(* Logix 5000 project; controller DIMTER vendor 1 type 14 code 77 rev 15.4; software revision 15.01; part 3 of 4 *)
(* tags used below, declared in another part *)
   ChainEjectorRunHourTimer : TIMER;   // Chain Ejector Run Hourmeter 1/10th Hour Timer
   CrossBelt1RunHourTimer : TIMER;   // Cross Belt 1 Run Hourmeter 1/10th Hour Timer
   CrossBelt2RunHourTimer : TIMER;   // Cross Belt 2 Run Hourmeter 1/10th Hour Timer
   CrossFeed1RunHourTimer : TIMER;   // Cross Feed 1 Run Hourmeter 1/10th Hour Timer
   CrossFeed2RunHourTimer : TIMER;   // Cross Feed 2 Run Hourmeter 1/10th Hour Timer
   DisplaySplashScreen : BOOL;
   F : BOOL[2016];   // Flags
   FlagTransferIndex : DINT;   // Index Register For Copying Flags to HMI Files
   FlagTransferIndex2 : DINT;
   FLASHER : TIMER;   // Lamp Flasher
   FLASHERB : TIMER;   // Lamp Flasher Reset
   RecordPieceSaw1 : BOOL;   // Record Piece Count For Shift Total
   RecordPieceSaw2 : BOOL;   // Record Piece Count For Shift Total
   Rollcase1RunHourTimer : TIMER;   // Rollcase 1 Run Hourmeter 1/10th Hour Timer
   Rollcase2RunHourTimer : TIMER;   // Rollcase 2 Run Hourmeter 1/10th Hour Timer
   Saw1RunHourTimer : TIMER;   // Saw 1 Run Hourmeter 1/10th Hour Timer
   Saw2RunHourTimer : TIMER;   // Saw 2 Run Hourmeter 1/10th Hour Timer
   SplashScreen : TIMER;
   T : TIMER[100];   // Timers
   WasteBelt1RunHourTimer : TIMER;   // Waste Belt 1 Run Hourmeter 1/10th Hour Timer
   WasteBelt2RunHourTimer : TIMER;   // Waste Belt 2 Run Hourmeter 1/10th Hour Timer
   A122 : ALIAS FOR Local:4:O.Data.2;   // O:4.0/2 A12.2 Reset Failure
   A123 : ALIAS FOR Local:4:O.Data.3;   // O:4.0/3 A12.3 Reset Buffer
   A143 : ALIAS FOR Local:5:O.Data.3;   // O:5.0/3 A143 Brake Cross Conveyor Front of Saw 1
   A144 : ALIAS FOR Local:5:O.Data.4;   // O:5.0/4 A144 Cross Feed 1 Fast Fwd
   A145 : ALIAS FOR Local:5:O.Data.5;   // O:5.0/5 A145 Cross Feed 1 Slow Fwd
   A147 : ALIAS FOR Local:5:O.Data.7;   // O:5.0/7 A147 Infeed Roller Saw 1
   A150 : ALIAS FOR Local:5:O.Data.8;   // O:5.0/8 A15.0 Rollcase 1 VSD Run Enable
   A151 : ALIAS FOR Local:5:O.Data.9;   // O:5.0/9 A15.1 Jog Rollcase 1 Set Speed
   A152 : ALIAS FOR Local:5:O.Data.10;   // O:5.0/10 A15.2 Forward Rotation Rollcase 1
   A153 : ALIAS FOR Local:5:O.Data.11;   // O:5.0/11 A15.3 Brake Rollcase Front of Saw 1
   A154 : ALIAS FOR Local:5:O.Data.12;   // O:5.0/12 A15.4 Rollcase 2 VSD Run Enable
   A155 : ALIAS FOR Local:5:O.Data.13;   // O:5.0/13 A155 Jog Rollcase 2 Set Speed
   A156 : ALIAS FOR Local:5:O.Data.14;   // O:5.0/14 A156 Forward Rotation Rollcase 2
   A157 : ALIAS FOR Local:5:O.Data.15;   // O:5.0/15 A157 Brake Rollcase 2
   A163 : ALIAS FOR Local:6:O.Data.3;   // O:6.0/3 A16.3 Brake Cross Conveyor Front of Saw 2
   A164 : ALIAS FOR Local:6:O.Data.4;   // O:6.0/4 A16.4 Cross Feed 2 Fast Fwd
   A165 : ALIAS FOR Local:6:O.Data.5;   // O:6.0/5 A16.5 Cross Feed 2 Slow Fwd
   A167 : ALIAS FOR Local:6:O.Data.7;   // O:6.0/7 A16.7 Infeed Roller Saw 2
   A172 : ALIAS FOR Local:6:O.Data.10;   // O:6.0/10 A17.2 Chain Ejector Brake
   A180 : ALIAS FOR Local:7:O.Data.0;   // O:7.0/0 A18.0 VSD Feed Contactor Rollcase 1
   A181 : ALIAS FOR Local:7:O.Data.1;   // O:7.0/1 A18.1 VSD Feed Contactor Rollcase 2
   A184 : ALIAS FOR Local:7:O.Data.4;   // O:7.0/4 A18.4 Waste Belt Conveyor 1
   A185 : ALIAS FOR Local:7:O.Data.5;   // O:7.0/5 A18.5 Waste Belt Conveyor 2
   A186 : ALIAS FOR Local:7:O.Data.6;   // O:7.0/6 A18.6 Cross Belt 1
   Debounce : TIMER[30];   // Debounce Timers
   Delay : TIMER[30];   // Delay Timers
   E00 : ALIAS FOR Local:1:I.Data.0;   // I:1.0/0 E0.0 Control Power On
   E01 : ALIAS FOR Local:1:I.Data.1;   // I:1.0/1 E0.1 Saw Hood 1 Closed
   E02 : ALIAS FOR Local:1:I.Data.2;   // I:1.0/2 E0.2 Saw Motor 1 On
   E03 : ALIAS FOR Local:1:I.Data.3;   // I:1.0/3 E0.3 Release - Feed Saw 1
   E06 : ALIAS FOR Local:1:I.Data.6;   // I:1.0/6 E0.6 Failure Conveyor in Front of Saw 1
   E07 : ALIAS FOR Local:1:I.Data.7;   // I:1.0/7 E0.7 Failure Conveyor in Front of Saw 2
   E11 : ALIAS FOR Local:1:I.Data.9;   // I:1.0/9 E1.1 Saw Hood 2 Closed
   E114 : ALIAS FOR Local:3:I.Data.28;   // I:3.1/12 E11.4 Transfer Station On
   E12 : ALIAS FOR Local:1:I.Data.10;   // I:1.0/10 E1.2 Saw Motor 2 On
   E13 : ALIAS FOR Local:1:I.Data.11;   // I:1.0/11 E1.3 Release - Feed Saw 2
   E22 : ALIAS FOR Local:1:I.Data.18;   // I:1.1/2 E2.2 Frequency Converter Rollcase in Front of Saw 1 Ready For Operation
   E23 : ALIAS FOR Local:1:I.Data.19;   // I:1.1/3 E2.3 Frequency Converter Rollcase in Front of Saw 2 Ready For Operation
   E27 : ALIAS FOR Local:1:I.Data.23;   // I:1.1/7 E2.7 Reset Safety Barrier at Transfer Station
   E32 : ALIAS FOR Local:1:I.Data.26;   // I:1.1/10 E3.2 Start Measurement Measurement Station
   E43 : ALIAS FOR Local:2:I.Data.3;   // I:2.0/3 E4.3 Infeed Saw 1 On
   E45 : ALIAS FOR Local:2:I.Data.5;   // I:2.0/5 E4.5 Transfer Station in Front of Saw On
   E46 : ALIAS FOR Local:2:I.Data.6;   // I:2.0/6 E4.6 Acknowledge Failure
   E53 : ALIAS FOR Local:2:I.Data.11;   // I:2.0/11 E5.3 Infeed Saw 2 On
   E54 : ALIAS FOR Local:2:I.Data.12;   // I:2.0/12 E5.4 Measuring Station On
   E55 : ALIAS FOR Local:2:I.Data.13;   // I:2.0/13 E5.5 Reset Defect Measuring Computer
   E56 : ALIAS FOR Local:2:I.Data.14;   // I:2.0/14 E5.6 Reset Buffer Measuring Computer
   E61 : ALIAS FOR Local:2:I.Data.17;   // I:2.1/1 E6.1 PE Infeed Saw 1
   E62 : ALIAS FOR Local:2:I.Data.18;   // I:2.1/2 E6.2 PE Front of Saw 1
   E63 : ALIAS FOR Local:2:I.Data.19;   // I:2.1/3 E6.3 PE Roller 1
   E64 : ALIAS FOR Local:2:I.Data.20;   // I:2.1/4 E6.4 Feed Saw 1 On
   E77 : ALIAS FOR Local:2:I.Data.31;   // I:2.1/15 E7.7 Cross Feed 1 at Front
   E81 : ALIAS FOR Local:3:I.Data.1;   // I:3.0/1 E8.1 PE Infeed Saw 2
   E82 : ALIAS FOR Local:3:I.Data.2;   // I:3.0/2 E8.2 PE Front of Saw 2
   E83 : ALIAS FOR Local:3:I.Data.3;   // I:3.0/3 E8.3 PE Roller 2
   E84 : ALIAS FOR Local:3:I.Data.4;   // I:3.0/4 E8.4 Feed Saw 2 On
   E97 : ALIAS FOR Local:3:I.Data.15;   // I:3.0/15 E9.7 Cross Feed 2 at Front
   FirstPass : BOOL;   // On for First Scan
   HMI_IntWords : INT[200];   // Integer Words to HMI
   HMI_RealWords : REAL[20];   // Real Words to HMI Transfer file
   Status : BOOL[224];   // Status Array
(* MainProgram, continued *)

ROUTINE HMI   (* ladder *)
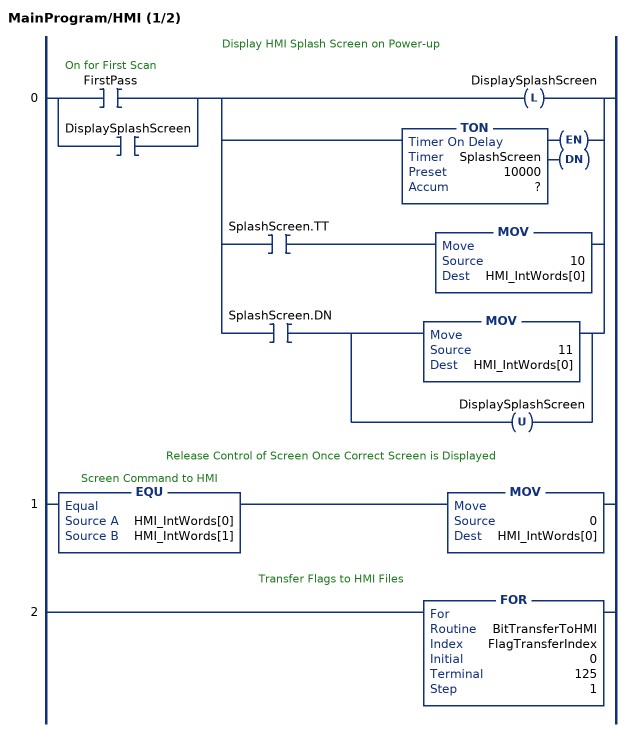
   // Display HMI Splash Screen on Power-up
   0: [XIC(FirstPass) ,XIC(DisplaySplashScreen) ][OTL(DisplaySplashScreen) ,TON(SplashScreen,?,?) ,XIC(SplashScreen.TT) MOV(10,HMI_IntWords[0]) ,XIC(SplashScreen.DN) [MOV(11,HMI_IntWords[0]) ,OTU(DisplaySplashScreen) ] ];
   // Release Control of Screen Once Correct Screen is Displayed
   1: EQU(HMI_IntWords[0],HMI_IntWords[1])MOV(0,HMI_IntWords[0]);
   // Transfer Flags to HMI Files
   2: FOR(BitTransferToHMI,FlagTransferIndex,0,125,1);
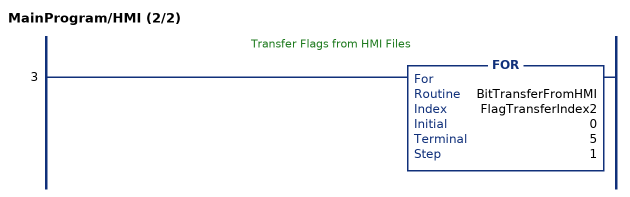
   // Transfer Flags from HMI Files
   3: FOR(BitTransferFromHMI,FlagTransferIndex2,0,5,1);
END_ROUTINE

ROUTINE MainRoutine   (* ladder *)
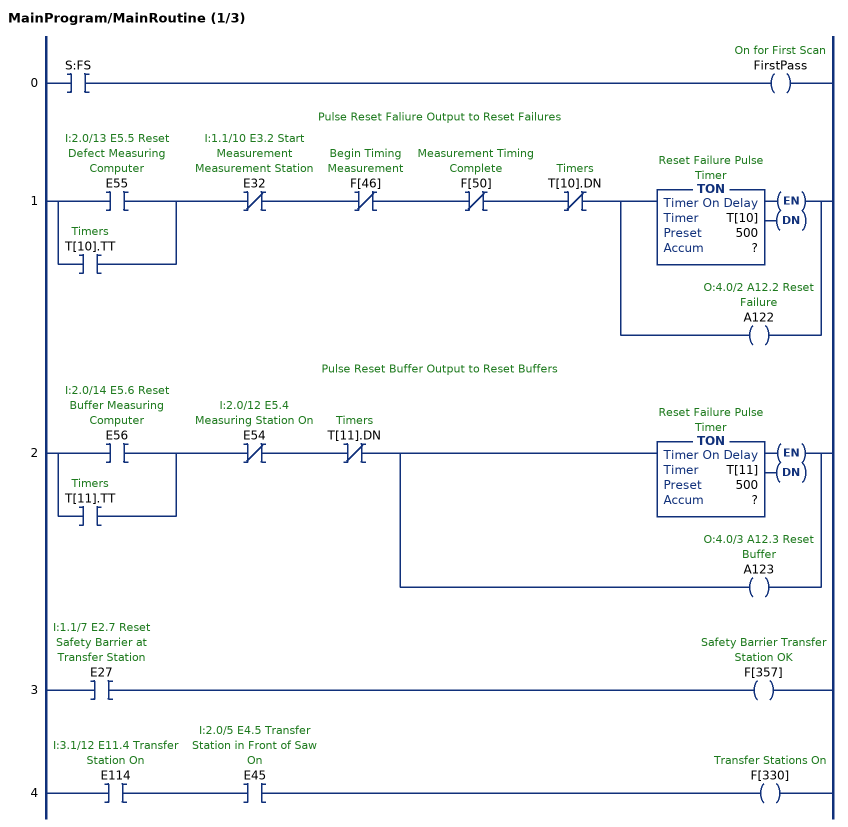
   0: XIC(S:FS)OTE(FirstPass);
   // Pulse Reset Faliure Output to Reset Failures
   1: [XIC(E55) ,XIC(T[10].TT) ]XIO(E32)XIO(F[46])XIO(F[50])XIO(T[10].DN)[TON(T[10],?,?) ,OTE(A122) ];
   // Pulse Reset Buffer Output to Reset Buffers
   2: [XIC(E56) ,XIC(T[11].TT) ]XIO(E54)XIO(T[11].DN)[TON(T[11],?,?) ,OTE(A123) ];
   3: XIC(E27)OTE(F[357]);
   4: XIC(E114)XIC(E45)OTE(F[330]);
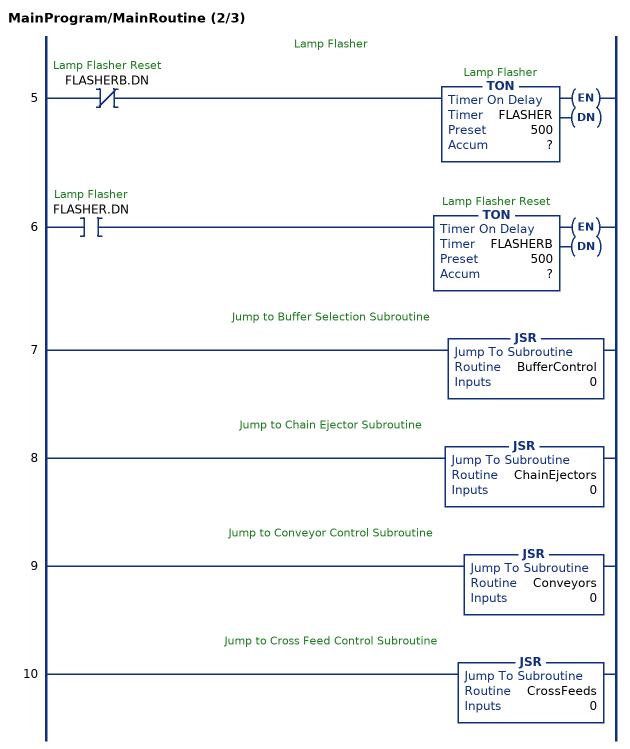
   // Lamp Flasher
   5: XIO(FLASHERB.DN)TON(FLASHER,?,?);
   6: XIC(FLASHER.DN)TON(FLASHERB,?,?);
   // Jump to Buffer Selection Subroutine
   7: JSR(BufferControl,0);
   // Jump to Chain Ejector Subroutine
   8: JSR(ChainEjectors,0);
   // Jump to Conveyor Control Subroutine
   9: JSR(Conveyors,0);
   // Jump to Cross Feed Control Subroutine
   10: JSR(CrossFeeds,0);
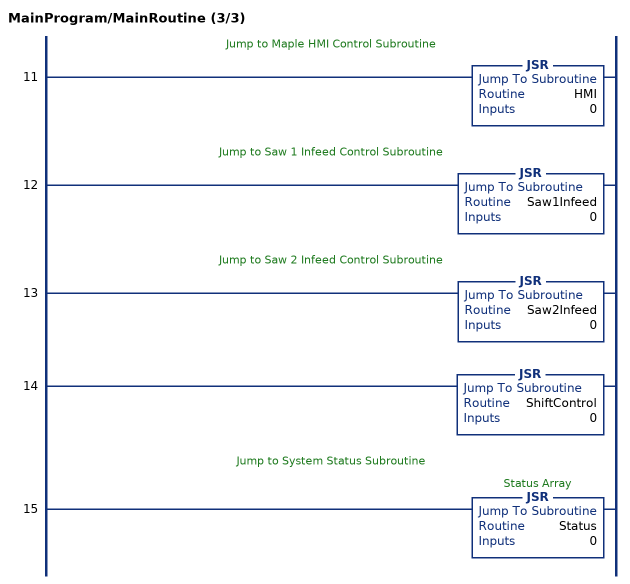
   // Jump to Maple HMI Control Subroutine
   11: JSR(HMI,0);
   // Jump to Saw 1 Infeed Control Subroutine
   12: JSR(Saw1Infeed,0);
   // Jump to Saw 2 Infeed Control Subroutine
   13: JSR(Saw2Infeed,0);
   14: JSR(ShiftControl,0);
   // Jump to System Status Subroutine
   15: JSR(Status,0);
END_ROUTINE

ROUTINE MotorRunCounters   (* ladder *)
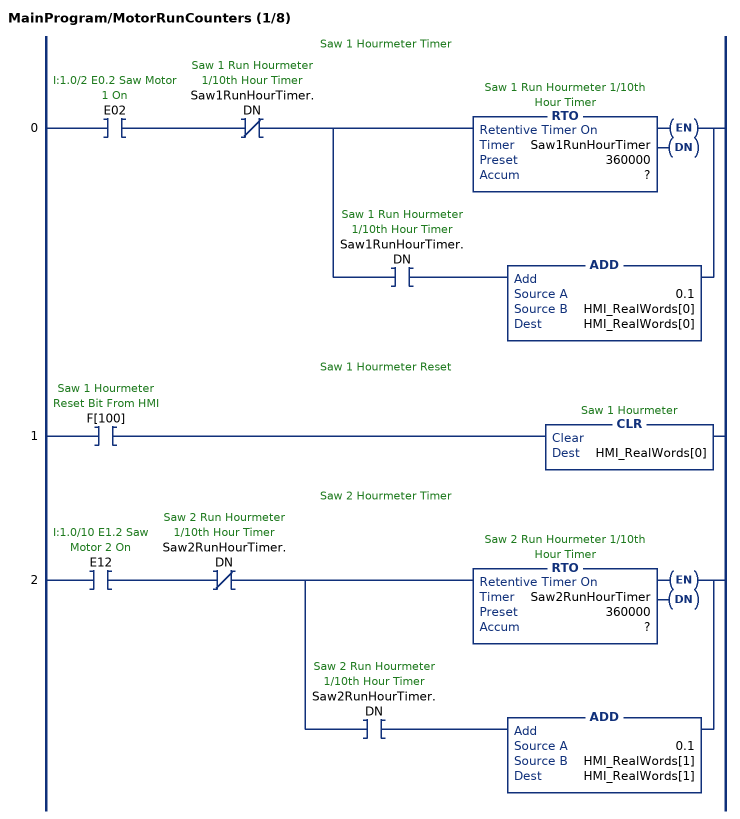
   // Saw 1 Hourmeter Timer
   0: XIC(E02)XIO(Saw1RunHourTimer.DN)[RTO(Saw1RunHourTimer,?,?) ,XIC(Saw1RunHourTimer.DN) ADD(0.1,HMI_RealWords[0],HMI_RealWords[0]) ];
   // Saw 1 Hourmeter Reset
   1: XIC(F[100])CLR(HMI_RealWords[0]);
   // Saw 2 Hourmeter Timer
   2: XIC(E12)XIO(Saw2RunHourTimer.DN)[RTO(Saw2RunHourTimer,?,?) ,XIC(Saw2RunHourTimer.DN) ADD(0.1,HMI_RealWords[1],HMI_RealWords[1]) ];
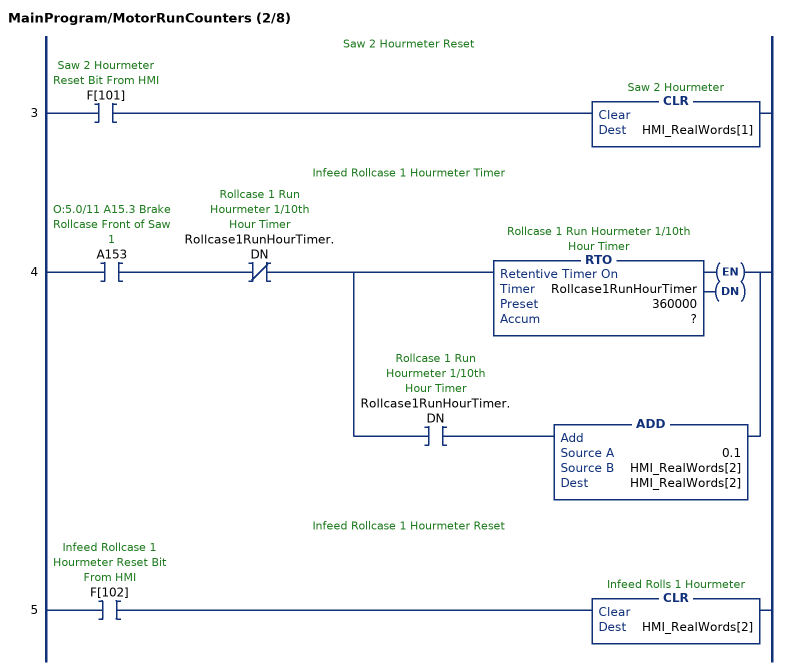
   // Saw 2 Hourmeter Reset
   3: XIC(F[101])CLR(HMI_RealWords[1]);
   // Infeed Rollcase 1 Hourmeter Timer
   4: XIC(A153)XIO(Rollcase1RunHourTimer.DN)[RTO(Rollcase1RunHourTimer,?,?) ,XIC(Rollcase1RunHourTimer.DN) ADD(0.1,HMI_RealWords[2],HMI_RealWords[2]) ];
   // Infeed Rollcase 1 Hourmeter Reset
   5: XIC(F[102])CLR(HMI_RealWords[2]);
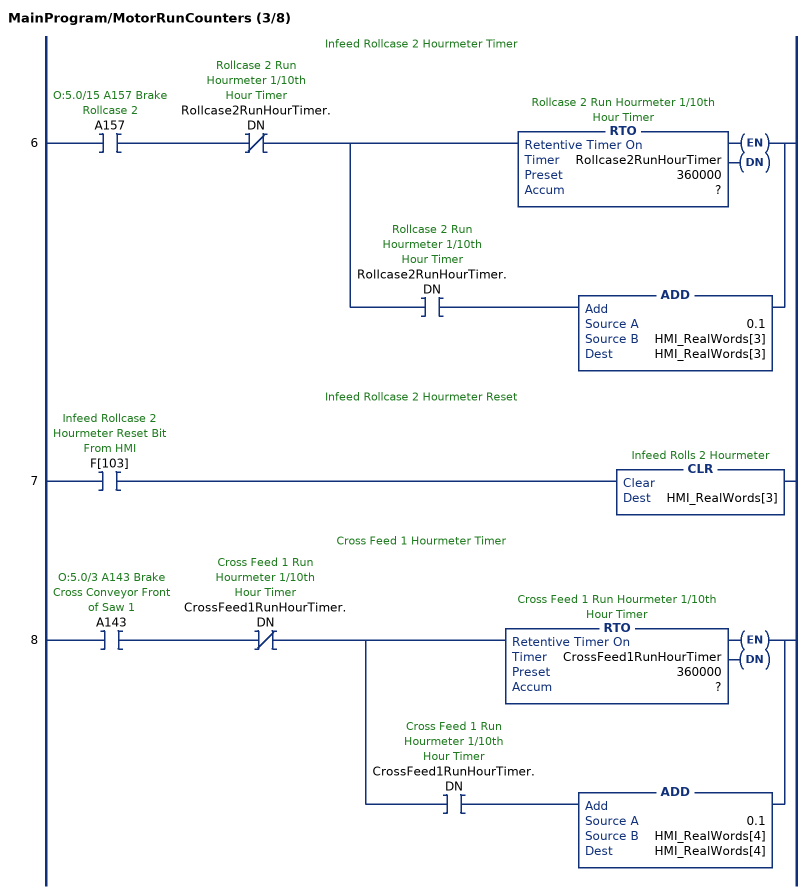
   // Infeed Rollcase 2 Hourmeter Timer
   6: XIC(A157)XIO(Rollcase2RunHourTimer.DN)[RTO(Rollcase2RunHourTimer,?,?) ,XIC(Rollcase2RunHourTimer.DN) ADD(0.1,HMI_RealWords[3],HMI_RealWords[3]) ];
   // Infeed Rollcase 2 Hourmeter Reset
   7: XIC(F[103])CLR(HMI_RealWords[3]);
   // Cross Feed 1 Hourmeter Timer
   8: XIC(A143)XIO(CrossFeed1RunHourTimer.DN)[RTO(CrossFeed1RunHourTimer,?,?) ,XIC(CrossFeed1RunHourTimer.DN) ADD(0.1,HMI_RealWords[4],HMI_RealWords[4]) ];
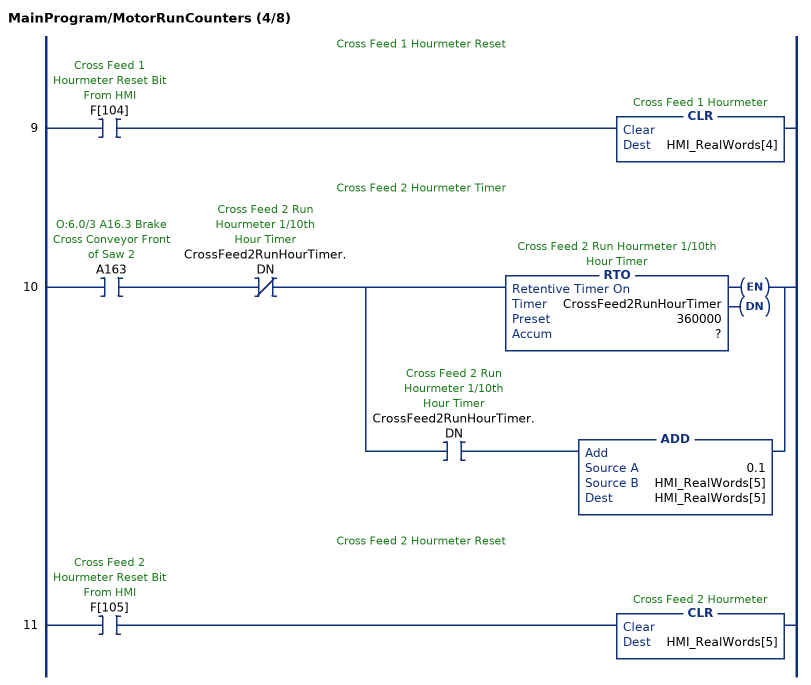
   // Cross Feed 1 Hourmeter Reset
   9: XIC(F[104])CLR(HMI_RealWords[4]);
   // Cross Feed 2 Hourmeter Timer
   10: XIC(A163)XIO(CrossFeed2RunHourTimer.DN)[RTO(CrossFeed2RunHourTimer,?,?) ,XIC(CrossFeed2RunHourTimer.DN) ADD(0.1,HMI_RealWords[5],HMI_RealWords[5]) ];
   // Cross Feed 2 Hourmeter Reset
   11: XIC(F[105])CLR(HMI_RealWords[5]);
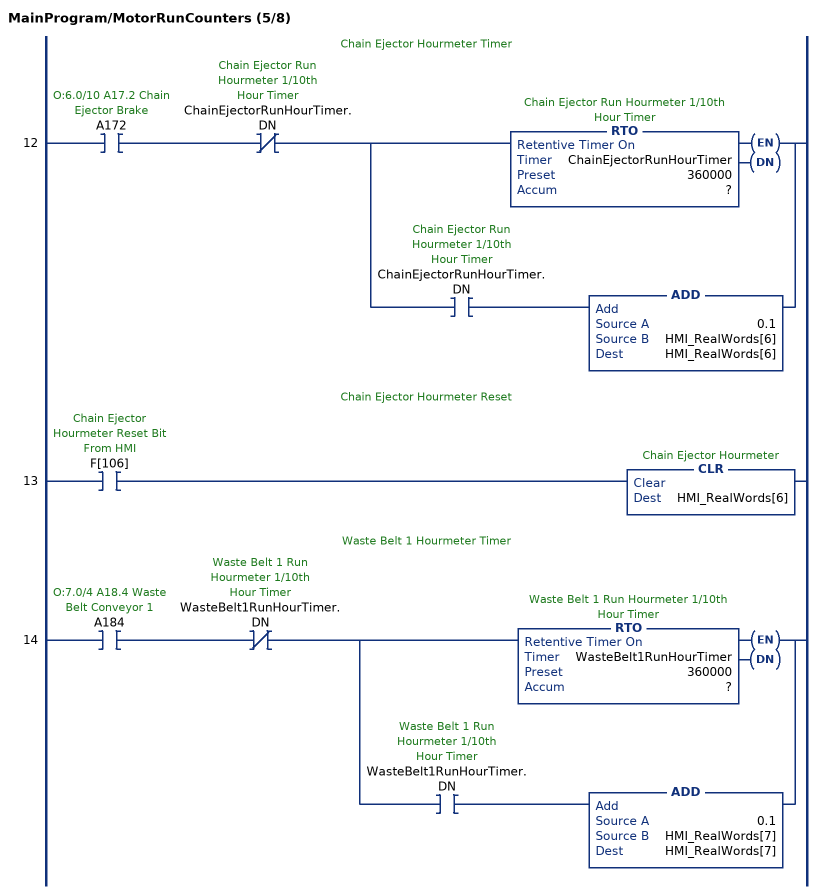
   // Chain Ejector Hourmeter Timer
   12: XIC(A172)XIO(ChainEjectorRunHourTimer.DN)[RTO(ChainEjectorRunHourTimer,?,?) ,XIC(ChainEjectorRunHourTimer.DN) ADD(0.1,HMI_RealWords[6],HMI_RealWords[6]) ];
   // Chain Ejector Hourmeter Reset
   13: XIC(F[106])CLR(HMI_RealWords[6]);
   // Waste Belt 1 Hourmeter Timer
   14: XIC(A184)XIO(WasteBelt1RunHourTimer.DN)[RTO(WasteBelt1RunHourTimer,?,?) ,XIC(WasteBelt1RunHourTimer.DN) ADD(0.1,HMI_RealWords[7],HMI_RealWords[7]) ];
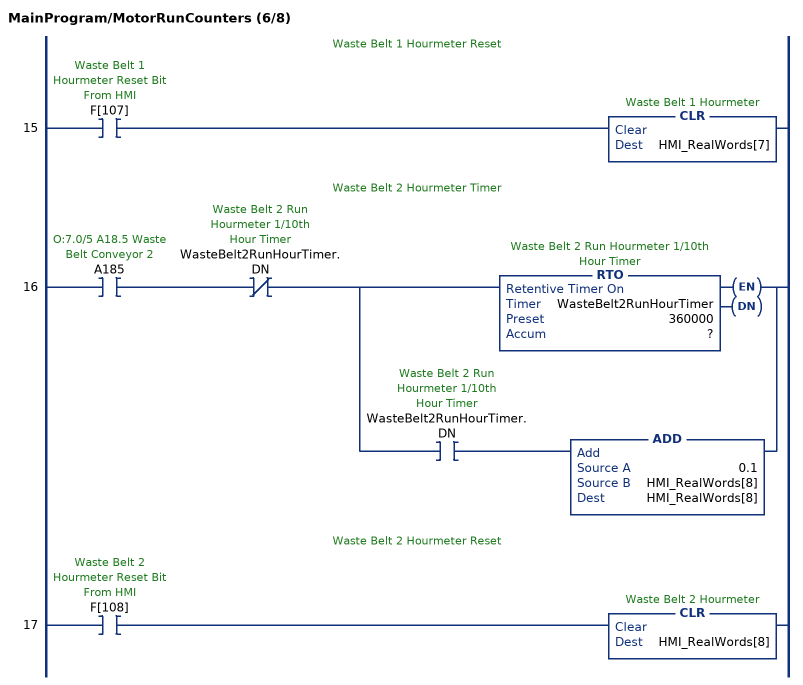
   // Waste Belt 1 Hourmeter Reset
   15: XIC(F[107])CLR(HMI_RealWords[7]);
   // Waste Belt 2 Hourmeter Timer
   16: XIC(A185)XIO(WasteBelt2RunHourTimer.DN)[RTO(WasteBelt2RunHourTimer,?,?) ,XIC(WasteBelt2RunHourTimer.DN) ADD(0.1,HMI_RealWords[8],HMI_RealWords[8]) ];
   // Waste Belt 2 Hourmeter Reset
   17: XIC(F[108])CLR(HMI_RealWords[8]);
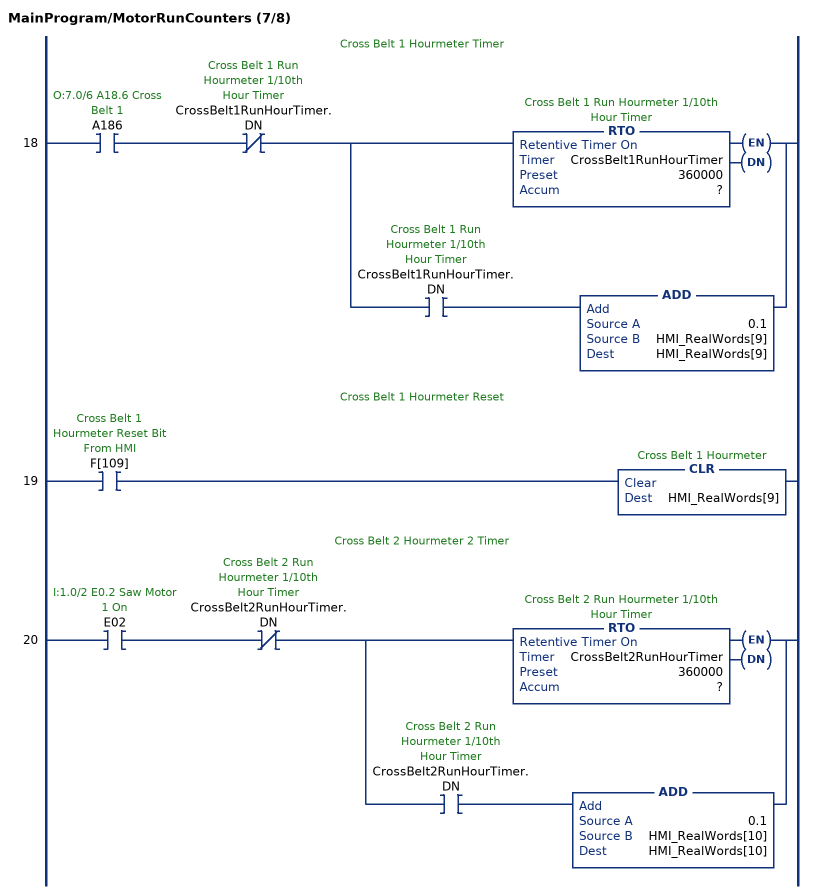
   // Cross Belt 1 Hourmeter Timer
   18: XIC(A186)XIO(CrossBelt1RunHourTimer.DN)[RTO(CrossBelt1RunHourTimer,?,?) ,XIC(CrossBelt1RunHourTimer.DN) ADD(0.1,HMI_RealWords[9],HMI_RealWords[9]) ];
   // Cross Belt 1 Hourmeter Reset
   19: XIC(F[109])CLR(HMI_RealWords[9]);
   // Cross Belt 2 Hourmeter 2 Timer
   20: XIC(E02)XIO(CrossBelt2RunHourTimer.DN)[RTO(CrossBelt2RunHourTimer,?,?) ,XIC(CrossBelt2RunHourTimer.DN) ADD(0.1,HMI_RealWords[10],HMI_RealWords[10]) ];
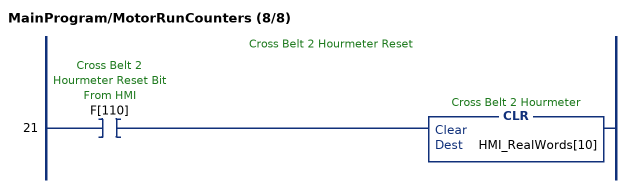
   // Cross Belt 2 Hourmeter Reset
   21: XIC(F[110])CLR(HMI_RealWords[10]);
END_ROUTINE

ROUTINE Saw1Infeed   (* ladder *)
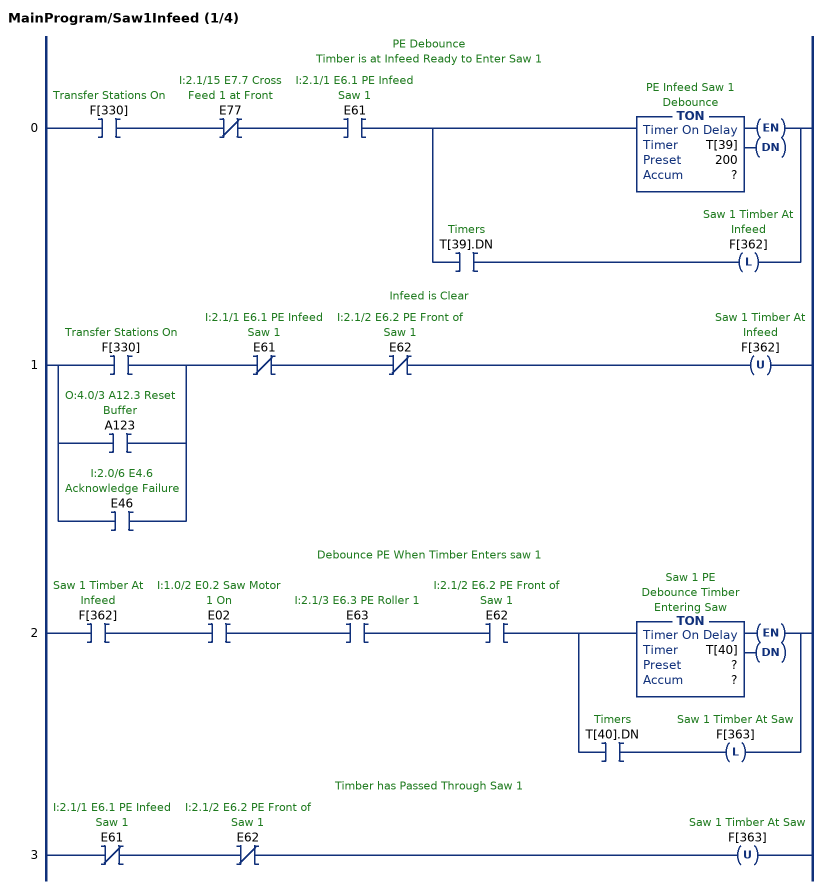
   // PE Debounce
   // Timber is at Infeed Ready to Enter Saw 1
   0: XIC(F[330])XIO(E77)XIC(E61)[TON(T[39],?,?) ,XIC(T[39].DN) OTL(F[362]) ];
   // Infeed is Clear
   1: [XIC(F[330]) ,XIC(A123) ,XIC(E46) ]XIO(E61)XIO(E62)OTU(F[362]);
   // Debounce PE When Timber Enters saw 1
   2: XIC(F[362])XIC(E02)XIC(E63)XIC(E62)[TON(T[40],?,?) ,XIC(T[40].DN) OTL(F[363]) ];
   // Timber has Passed Through Saw 1
   3: XIO(E61)XIO(E62)OTU(F[363]);
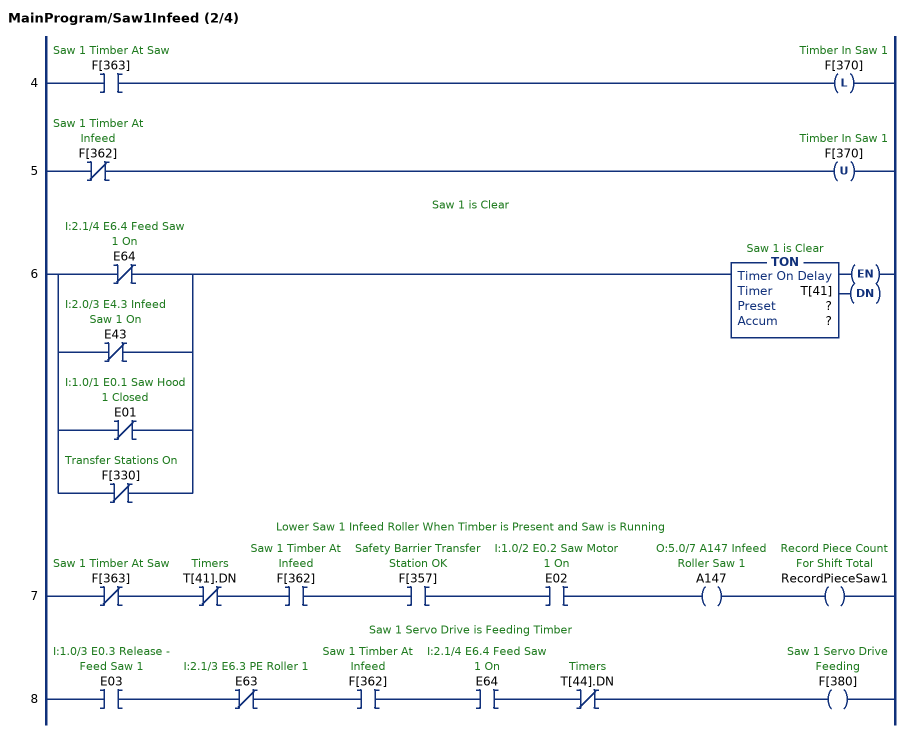
   4: XIC(F[363])OTL(F[370]);
   5: XIO(F[362])OTU(F[370]);
   // Saw 1 is Clear
   6: [XIO(E64) ,XIO(E43) ,XIO(E01) ,XIO(F[330]) ]TON(T[41],?,?);
   // Lower Saw 1 Infeed Roller When Timber is Present and Saw is Running
   7: XIO(F[363])XIO(T[41].DN)XIC(F[362])XIC(F[357])XIC(E02)OTE(A147)OTE(RecordPieceSaw1);
   // Saw 1 Servo Drive is Feeding Timber
   8: XIC(E03)XIO(E63)XIC(F[362])XIC(E64)XIO(T[44].DN)OTE(F[380]);
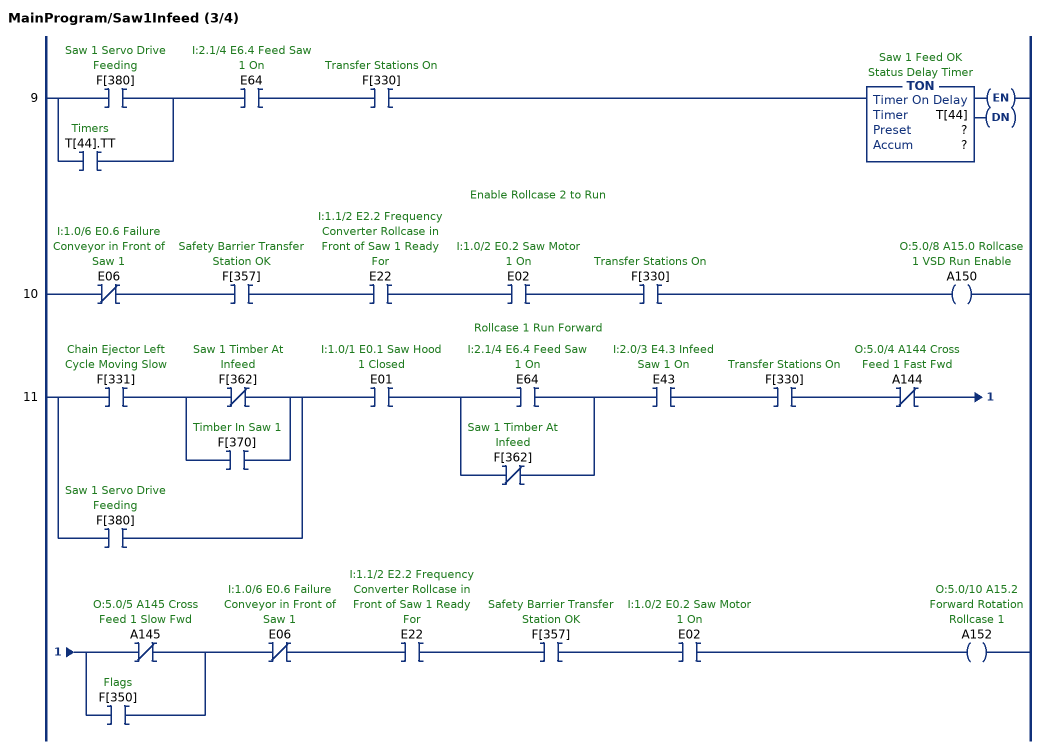
   9: [XIC(F[380]) ,XIC(T[44].TT) ]XIC(E64)XIC(F[330])TON(T[44],?,?);
   // Enable Rollcase 2 to Run
   10: XIO(E06)XIC(F[357])XIC(E22)XIC(E02)XIC(F[330])OTE(A150);
   // Rollcase 1 Run Forward
   11: [XIC(F[331]) [XIO(F[362]) ,XIC(F[370]) ] ,XIC(F[380]) ]XIC(E01)[XIC(E64) ,XIO(F[362]) ]XIC(E43)XIC(F[330])XIO(A144)[XIO(A145) ,XIC(F[350]) ]XIO(E06)XIC(E22)XIC(F[357])XIC(E02)OTE(A152);
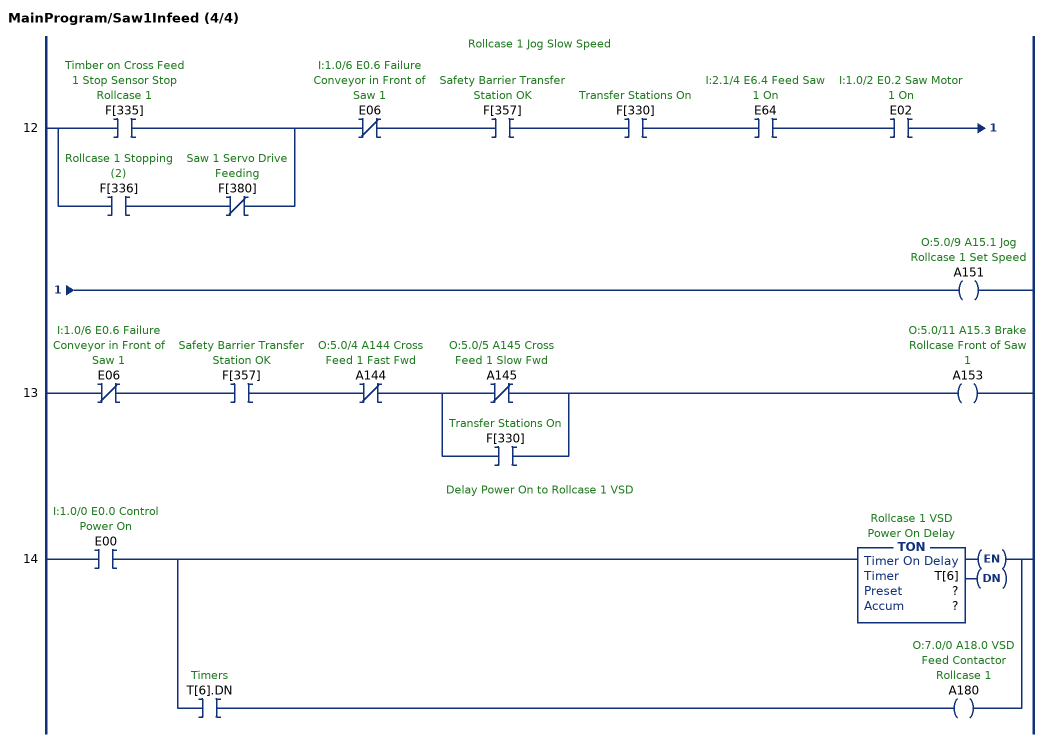
   // Rollcase 1 Jog Slow Speed
   12: [XIC(F[335]) ,XIC(F[336]) XIO(F[380]) ]XIO(E06)XIC(F[357])XIC(F[330])XIC(E64)XIC(E02)OTE(A151);
   13: XIO(E06)XIC(F[357])XIO(A144)[XIO(A145) ,XIC(F[330]) ]OTE(A153);
   // Delay Power On to Rollcase 1 VSD
   14: XIC(E00)[TON(T[6],?,?) ,XIC(T[6].DN) OTE(A180) ];
END_ROUTINE

ROUTINE Saw2Infeed   (* ladder *)
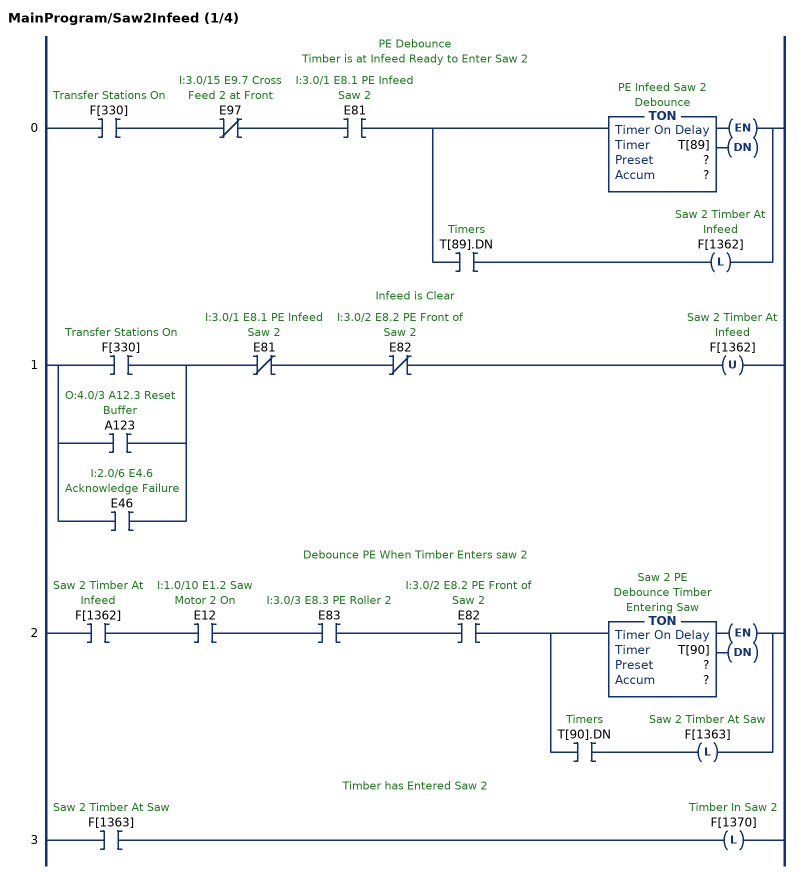
   // PE Debounce
   // Timber is at Infeed Ready to Enter Saw 2
   0: XIC(F[330])XIO(E97)XIC(E81)[TON(T[89],?,?) ,XIC(T[89].DN) OTL(F[1362]) ];
   // Infeed is Clear
   1: [XIC(F[330]) ,XIC(A123) ,XIC(E46) ]XIO(E81)XIO(E82)OTU(F[1362]);
   // Debounce PE When Timber Enters saw 2
   2: XIC(F[1362])XIC(E12)XIC(E83)XIC(E82)[TON(T[90],?,?) ,XIC(T[90].DN) OTL(F[1363]) ];
   // Timber has Entered Saw 2
   3: XIC(F[1363])OTL(F[1370]);
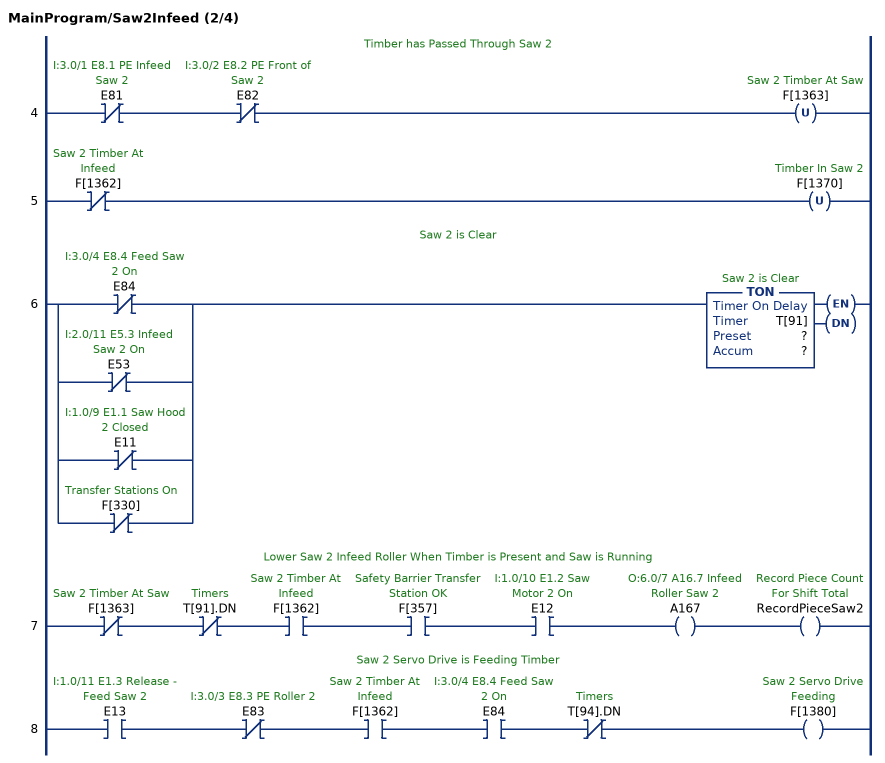
   // Timber has Passed Through Saw 2
   4: XIO(E81)XIO(E82)OTU(F[1363]);
   5: XIO(F[1362])OTU(F[1370]);
   // Saw 2 is Clear
   6: [XIO(E84) ,XIO(E53) ,XIO(E11) ,XIO(F[330]) ]TON(T[91],?,?);
   // Lower Saw 2 Infeed Roller When Timber is Present and Saw is Running
   7: XIO(F[1363])XIO(T[91].DN)XIC(F[1362])XIC(F[357])XIC(E12)OTE(A167)OTE(RecordPieceSaw2);
   // Saw 2 Servo Drive is Feeding Timber
   8: XIC(E13)XIO(E83)XIC(F[1362])XIC(E84)XIO(T[94].DN)OTE(F[1380]);
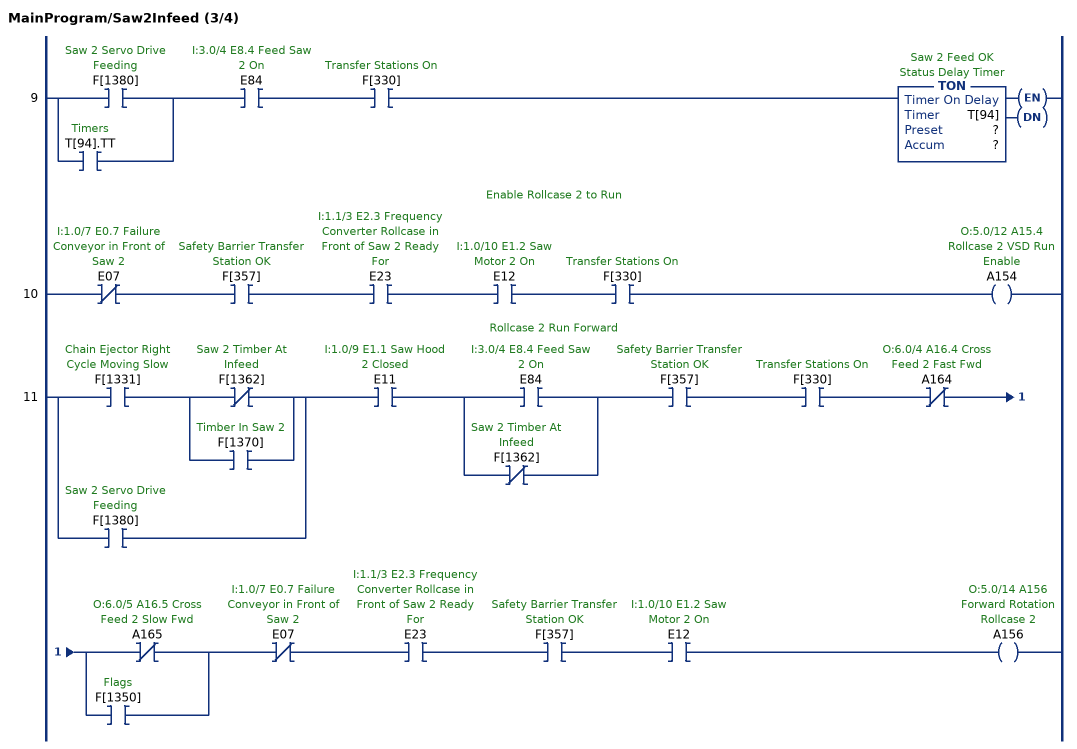
   9: [XIC(F[1380]) ,XIC(T[94].TT) ]XIC(E84)XIC(F[330])TON(T[94],?,?);
   // Enable Rollcase 2 to Run
   10: XIO(E07)XIC(F[357])XIC(E23)XIC(E12)XIC(F[330])OTE(A154);
   // Rollcase 2 Run Forward
   11: [XIC(F[1331]) [XIO(F[1362]) ,XIC(F[1370]) ] ,XIC(F[1380]) ]XIC(E11)[XIC(E84) ,XIO(F[1362]) ]XIC(F[357])XIC(F[330])XIO(A164)[XIO(A165) ,XIC(F[1350]) ]XIO(E07)XIC(E23)XIC(F[357])XIC(E12)OTE(A156);
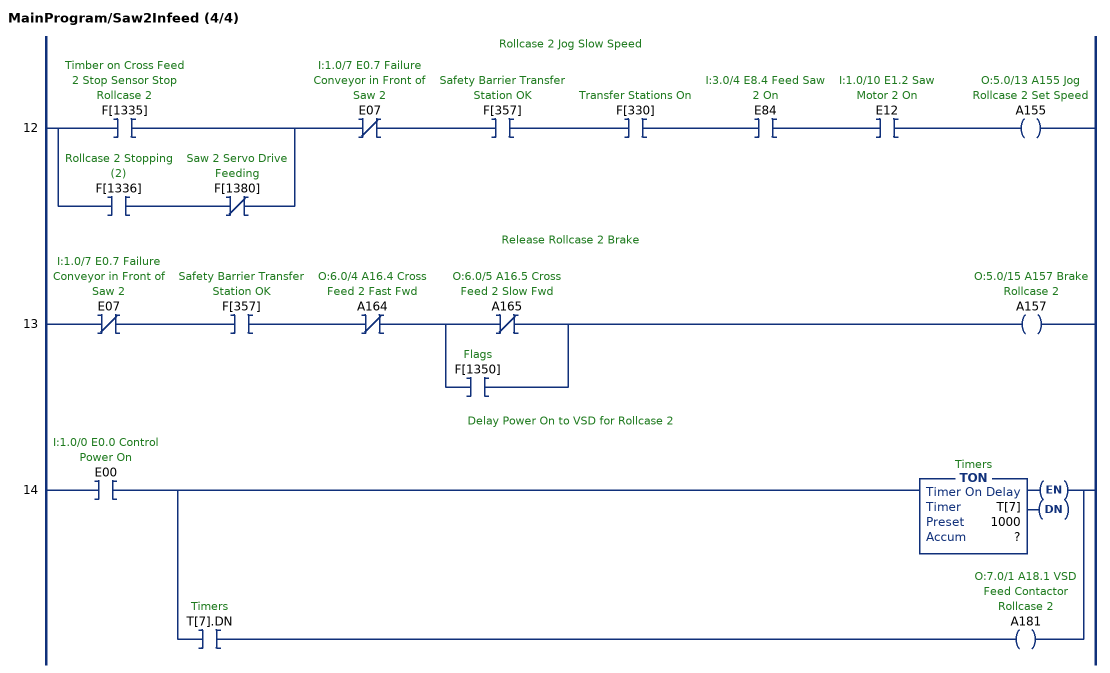
   // Rollcase 2 Jog Slow Speed
   12: [XIC(F[1335]) ,XIC(F[1336]) XIO(F[1380]) ]XIO(E07)XIC(F[357])XIC(F[330])XIC(E84)XIC(E12)OTE(A155);
   // Release Rollcase 2 Brake
   13: XIO(E07)XIC(F[357])XIO(A164)[XIO(A165) ,XIC(F[1350]) ]OTE(A157);
   // Delay Power On to VSD for Rollcase 2
   14: XIC(E00)[TON(T[7],?,?) ,XIC(T[7].DN) OTE(A181) ];
END_ROUTINE
